(* Logix 5000 project; controller Transcat vendor 1 type 14 code 152 rev 32.11; software revision 32.02 *)

TASK MainTask (continuous, watchdog 500 ms) : MainProgram

MODULES
   Local : vendor 1 type 14 code 152 (PointIO 0, rev 32.11)
      MX201_LowerHowesVFD : PowerFlex 525-EENET (Ethernet 192.168.1.192, rev 5.1, Output RPI 20 ms)   // VFD for Lower Howes Mixer
           MX201_LowerHowesVFD:I.Ready   // LowerHowes Drive Ready Status
           MX201_LowerHowesVFD:I.Faulted   // LowerHowes Drive Faulted
           MX201_LowerHowesVFD:I.Active   // LowerHowes Drive Active
           MX201_LowerHowesVFD:O.Stop   // Drive Stop
      MX101_UpperHowesVFD : PowerFlex 525-EENET (Ethernet 192.168.1.191, rev 5.1, Output RPI 20 ms)   // VFD for Upper Howes Mixer
           MX101_UpperHowesVFD:I.Faulted   // UpperHowes Drive Faulted
           MX101_UpperHowesVFD:I.Active   // UpperHowes Drive Active
           MX101_UpperHowesVFD:I.Ready   // UpperHowes Drive Ready Status
           MX101_UpperHowesVFD:O.FreqCommand   // Input Hz into Source A: 0-60 Hz range
           MX101_UpperHowesVFD:O.Stop   // Drive Stop
           MX101_UpperHowesVFD:O.Start   // Drive Start
      VF101_Medium_Feeder : PowerFlex 525-EENET (Ethernet 192.168.1.193, rev 5.1, Output RPI 20 ms)   // Medium Feeder
      VF201_Small_Feeder_2 : PowerFlex 525-EENET (Ethernet 192.168.1.194, rev 5.1, Output RPI 20 ms)   // Small Feeder 2
      Thayer1_BS : ETHERNET-MODULE (Ethernet 192.168.1.140, rev 1.1, Output RPI 50 ms)   // Thayer 1 Weight Belt Feeder
      SBC2000_1_Acrison : ETHERNET-MODULE (Ethernet 192.168.1.150, rev 1.1, Output RPI 250 ms)   // Acrison Drive 1 to control Small Feeder 1
           SBC2000_1_Acrison:I.Data[1]   // PV - Feedrate - kg/hr
           SBC2000_1_Acrison:I.Data[2]   // Totalizer 1 - kg
           SBC2000_1_Acrison:I.Data[4]   // Hopper Level - %
           SBC2000_1_Acrison:I.Data[3]   // OT - Motor Speed - %
           SBC2000_1_Acrison:I.Data   // Ethernet Input Array
           SBC2000_1_Acrison:I.Data[0]   // SP-FeedRate - kg/hr
           SBC2000_1_Acrison:O.Data[15]   // When Command_Bits is 1, machine is running.
      Thayer2_BS : ETHERNET-MODULE (Ethernet 192.168.1.160, rev 1.1, Output RPI 50 ms)   // Thayer 2 Weigh Belt Feeder
      AENTPointIO : 1734-AENT (Ethernet 192.168.1.190, rev 3.1, Output RPI 20 ms)
         Slot1_420_8Input : vendor 1 type 115 code 210 (PointIO 1, rev 3.1, Input RPI 80 ms)
              AENTPointIO:1:I.Ch0Data   // LowerHowesSpeedSensorSignal
         Slot2_24V_8DI : 1734-IB8 (PointIO 2, rev 3.1)
      Discrete_IO : Embedded (PointIO 1, rev 32.11, Output RPI 20 ms)
           Local:1:O.Data.0   // Red Beacon Light
           Local:1:O.Data.3   // Blue Beacon Light
           Local:1:O.Data.1   // Yellow Beacon Light
           Local:1:O.Data.2   // Green Beacon Light
           Local:1:O.Data.4   // Beacon Buzzer/Sound
END_MODULES

TYPE Acrison_Feeder :   // Acrison Feeder Tags
STRUCT
   AutoMan : BOOL;   // On - Auto Control - follows AutoRun bit, Off - Manaul Control - follows Manual Run bit
   ManualRun : BOOL;   // On - Runs feeder in Manual, Off - Stops feeder in manual
   AutoRun : BOOL;   // On - Runs feeder in Auto Off - Stops feeder in Auto
   Interlock : BOOL;   // Interlock bit - if on - Feeder will not run
   Output : BOOL;   // On - Feeder runs, Off Feeder stops
   Int_Status : DINT;   // 32 Status bits from feeder
   SP_HMI : REAL;   // setpoint from HMI
   SP_READ : REAL;   // setpoint read back from controller
   Enable : BOOL;   // Enable logic to run feeder
   OT_Actual_Hz : REAL;   // The current output of the VFD in Hz
   FreqHz_Real : REAL;   // The command frequency of the drive in Hz
   CycleTime : TIMER;   // running time of current cycle
   CampTime : TIMER;   // running time of current campaign / batch
   TotalTime : TIMER;   // total time the device / motor has run since last reset
   OneShots : BOOL[32];   // 32 Booleans to hold one-shots assicated with this device
   TimeRunTarget : DINT;   // Target Amount of time in seconds to run the device
   StartDelay : TIMER;   // Delay before motor start
   StartDelayms : DINT;   // Start delay in milliseconds
   TimeRunStart : BOOL;   // Bit to start and run a timed run
END_STRUCT
END_TYPE

TYPE BronkhorstFlowMeter :   // Read and write values for Bronkhorst Flow Meters
STRUCT
   SP_R : REAL;   // Set Point - FlowRate - Read - g/min - read from Flow Meter
   PV_R : REAL;   // Process Variable - FlowRate - Read - g/min
   OT_R : REAL;   // Output - PumpSpeed - Read - %
   TempC : REAL;   // Temperaure - Read - Deg C
   Density : REAL;   // Density - Read - g/liter
   Usertag : STRING;   // User Tag in Flow Meter - String
   FBNode : INT;   // Flow Bus Node # - Integer
   Model : STRING;   // Flow Meter Model #
   Serial : STRING;   // Flow Meter Serial #
   Capacity : REAL;   // Max Flow Rate of Flow Meter
   Enable : BOOL;   // Device enable bit
   AutoMan : BOOL;   // Select Auto / Manual Mode
   AutoRun : BOOL;   // On / Off in Auto Mode
   ManualRun : BOOL;   // On / Off- in Manual Mode
   Interlock : BOOL;   // Interlock Bit
   Output : BOOL;   // Output Bit for Device
   SP_HMI : REAL;   // Setpoint from HMI
   SP_W : REAL;   // Setpoint - flowrate g/min - write to Flow Meter from PLC
   Connected : BOOL;   // Is flow meter connecte to the flow bus network
   Alarm : BOOL;   // Alarm Bit - if on flow meter in ALarm Status
   Running : BOOL;   // the flow meter is running / dosing
   AlarmReset : BOOL;   // bit to toggle to reset alarm
   AlarmID : INT;   // Integer # that describes the type of Alarm
   ReadTime : INT;   // time in milliseconds to read the flow meter data
   DevPct : REAL;   // % deviation of process variable from setpoint
   CycleTime : TIMER;   // running time of current cycle
   CampTime : TIMER;   // running time of current campaign
   TotalTime : TIMER;   // total time the device / motor has run since last reset
   OneShots : BOOL[32];   // 32 Booleans to hold one-shots assicated with this device
   TimeRunTarget : DINT;   // Target Amount of time in seconds to run the device
   StartDelay : TIMER;   // Delay before motor start
   StartDelayms : DINT;   // Start delay in milliseconds
   TimeRunStart : BOOL;   // Bit to start and run a timed run
   Totalizer : REAL;   // Total dosed by flow meter since last reset
   TotalizerReset : BOOL;   // Bit to reset the totalizer (called a counter in Bronkhorst literature)
END_STRUCT
END_TYPE

TYPE Howes_Mixer :   // Howes Mixer Tags
STRUCT
   AutoMan : BOOL;   // On - Auto Control - follows AutoRun bit, Off - Manaul Control - follows Manual Run bit
   ManualRun : BOOL;   // On - Runs feeder in Manual, Off - Stops feeder in manual
   AutoRun : BOOL;   // On - Runs feeder in Auto Off - Stops feeder in Auto
   Interlock : BOOL;   // Interlock bit - if on - Feeder will not run
   Output : BOOL;   // On - Feeder runs, Off Feeder stops
   Int_Status : DINT;   // 32 Status bits from feeder
   SP_HMI : REAL;   // setpoint from HMI
   SP_READ : REAL;   // setpoint read back from controller
   Enable : BOOL;   // Enable logic to run mixer
   FreqHz_Real : REAL;   // Frequency in Hz expressed as real #
   OT_Actual_Hz : REAL;   // The current output of the drive in Hz
   CycleTime : TIMER;   // currnet cycle run time
   CampTime : TIMER;   // current campaign run time
   TotalTime : TIMER;   // total run time since last reset
   OneShots : BOOL[32];   // 32 Booleans to hold one shots associated with this device
   TimeRunTarget : DINT;   // Target Amount of time in seconds to run the device
   TimeRunStart : BOOL;   // Bit to start and run a timed run
   StartDelay : TIMER;   // Delay before motor starts
   StartDelayms : DINT;   // Delay before motor starts in milliseconds
   RPM : REAL;   // RPM from speed sensor
END_STRUCT
END_TYPE

TYPE Thayer_WB_Feeder :   // Thayer WB Feeder Tags
STRUCT
   AutoMan : BOOL;   // On - Auto Control - follows AutoRun bit, Off - Manaul Control - follows Manual Run bit
   ManualRun : BOOL;   // On - Runs feeder in Manual, Off - Stops feeder in manual
   AutoRun : BOOL;   // On - Runs feeder in Auto Off - Stops feeder in Auto
   Interlock : BOOL;   // Interlock bit - if on - Feeder will not run
   Output : BOOL;   // On - Feeder runs, Off Feeder stops
   Int_Status : DINT;   // 32 Status bits from feeder
   SP_HMI : REAL;   // setpoint from HMI
   SP_READ : REAL;   // setpoint read back from controller
   Enable : BOOL;   // Enable logic to run feeder
   CycleTime : TIMER;   // current cycle run time
   CampTime : TIMER;   // current campaing run time
   TotalTime : TIMER;   // total run time since last reset
   OneShots : BOOL[32];   // 32 Booleans to hold one-shots assicated with this device
   TimeRunTarget : DINT;   // Target Amount of time in seconds to run the device - from recipe
   StartDelay : TIMER;   // Delay before starting motor / equipment
   StartDelayms : DINT;   // Start delay in milliseconds
   TimeRunStart : BOOL;   // Bit to start and run a timed run
END_STRUCT
END_TYPE

VAR_GLOBAL   (* controller tags *)
   AcrisonFeedRateSetPoint : MESSAGE;   // Message Command to Write to Feed Rate Set Point in Acrison from GF103.SP_HMI in kg/hr
        MessageParameters(ServiceCode := 16#0010, LocalElement := GF301.SP_HMI, ...)
   alwaysOFF : BOOL;
   BeaconBeepAlarm : ALIAS FOR Local:1:O.Data.4;   // Beep Alarm
   BeaconBlueLight : ALIAS FOR Local:1:O.Data.3;   // Blue Beacon Light
   BeaconGreenLight : ALIAS FOR Local:1:O.Data.2;   // Green Beacon Light
   BeaconRedLight : ALIAS FOR Local:1:O.Data.0;   // Red Beacon Light
   BeaconYellowLight : ALIAS FOR Local:1:O.Data.1;   // Yellow Beacon Light
   Beep : BOOL;   // Bit to Activte Beacon Alarm
   FT103 : BronkhorstFlowMeter := (PV_R := 8.803709, TempC := 22.585506, Density := 9999.0, Usertag := 'FT-103', Model := 'M55-RGD-25-0-S', Serial := 'M22213015A', Capacity := 1000.00006, Enable := 1, SP_HMI := 100.0, Connected := 1, ReadTime := 136, CycleTime.PRE := 288000000, CycleTime.ACC := 19487, CampTime.PRE := 28800000, CampTime.ACC := 10001, TotalTime.PRE := 999999999, TotalTime.ACC := 114629, Totalizer := 30.49);
   FT104 : BronkhorstFlowMeter := (PV_R := -9.60369, TempC := 22.258062, Density := 9999.0, Usertag := 'FT-104          ', Model := 'M55-RGD-25-0-S', Serial := 'M22213015C', Capacity := 10000.0, Enable := 1, SP_HMI := 100.0, Connected := 1, ReadTime := 80, CycleTime.PRE := 288000000, CycleTime.ACC := 3248, CampTime.PRE := 28800000, CampTime.ACC := 10001, TotalTime.PRE := 999999999, TotalTime.ACC := 84417, StartDelay.PRE := 2000, StartDelayms := 2, Totalizer := 6.64);
   FT105 : BronkhorstFlowMeter := (PV_R := 0.5630569, TempC := 29.962246, Density := 5.6385093, Usertag := 'FT-105          ', Model := 'M14-RGD-22-0-S', Serial := 'M20210127A', Capacity := 202.79999, Enable := 1, SP_HMI := 12.5, Connected := 1, ReadTime := 63, CycleTime.PRE := 288000000, CycleTime.ACC := 11357, CampTime.PRE := 28800000, CampTime.ACC := 10001, TotalTime.PRE := 999999999, TotalTime.ACC := 55929, StartDelay.PRE := 4000, StartDelayms := 4, Totalizer := 1840865.0);
   GF101 : Thayer_WB_Feeder := (SP_HMI := 10.0, SP_READ := 10.0, Enable := 1, CycleTime.PRE := 288000000, CycleTime.ACC := 9195, CampTime.PRE := 28800000, CampTime.ACC := 10001, TotalTime.PRE := 999999999, TotalTime.ACC := 1761327, StartDelay.PRE := 2000, StartDelayms := 2);   // Thayer 1 Tags
   GF101_Alarm_ExcessDevSP : ALIAS FOR Thayer1_BS:I.Data[8].7;   // Thayer 1 (GF101) - Alarm - excessive deviation from SP
   GF101_LoadCell : ALIAS FOR Thayer1Data[15];   // Thayer 1 (GF101) load cell in lbs
   GF101_LoadCellTempF : ALIAS FOR Thayer1Data[16];   // Thayer 1 (GF101) load cell temperature in Deg F
   GF101_OutputPct : ALIAS FOR Thayer1Data[5];   // Thayer 1 (GF101) Output to motor in pct - raw
   GF101_RunningLoad : ALIAS FOR Thayer1Data[0];   // Thayer 1 (GF101) Running Load - current load on belt in lbs
   GF101_RunningRate : ALIAS FOR Thayer1Data[1];   // Thayer 1 (GF101) Running Rate - current PV displayed on the operator screen
   GF101_RunningSpeed : ALIAS FOR Thayer1Data[2];   // Thayer 1 (GF101) Running Soeed - current speed of the belt in ft/min?
   GF101_SetPoint : ALIAS FOR Thayer1Data[3];   // Thayer 1 (GF101) SetPoint - in lb/min
   GF101_Shutdown_ExcessDevSp : ALIAS FOR Thayer1_BS:I.Data[10].7;   // Thayer 1 (GF101) - Shutdown - excessive deviation from SP
   GF101_Status_AutoMan : ALIAS FOR Thayer1_BS:I.Data[0].1;   // Thayer 1 (GF101) - Auto / Manual Status - 1 = Auto 0 = Manual
   GF101_Status_Coasting : ALIAS FOR Thayer1_BS:I.Data[0].2;   // Thayer 1 (GF101) - Coasting to stop of shutdown - 1 = Coasting, 0 = Not coasting
   GF101_Status_EchoBack : ALIAS FOR Thayer1_BS:I.Data[0].13;   // Thayer 1 (GF101) - Echo back bit
   GF101_Status_HeartBeat : ALIAS FOR Thayer1_BS:I.Data[0].14;   // Thayer 1 (GF101) - HeartBeat - every 5 seconds
   GF101_Status_Interlocked : ALIAS FOR Thayer1_BS:I.Data[0].8;   // Thayer 1 (GF101) - Interlocked Bit - 1 = Interlocked 0 = Not Interlocked
   GF101_Status_RunStop : ALIAS FOR Thayer1_BS:I.Data[0].0;   // Thayer 1 (GF101) - Operating Status - 1 = Running 0 = Stopped
   GF101_Status_TachGT0 : ALIAS FOR Thayer1_BS:I.Data[0].9;   // Thayer 1 (GF101) - 1 = Tachometer > 0 0 = Tachometer = 0
   GF101_TachHz : ALIAS FOR Thayer1Data[14];   // Thayer 1 (GF101) Tachometer in Hz
   GF101_Totalizer1 : ALIAS FOR Thayer1Data[9];   // Thayer 1 (GF101) Totalizer 1 in lbs
   GF101_Totalizer2 : ALIAS FOR Thayer1Data[10];   // Thayer 1 (GF101) Totalizer 2 in lbs
   GF101_Write_Acknowledge : ALIAS FOR Thayer1_BS:O.Data[2].5;   // Thayer 1 (GF101) Acknowledge
   GF101_Write_AutoMan : ALIAS FOR Thayer1_BS:O.Data[0].1;   // Thayer 1 (GF101) Auto / Manual 1 = Auto 2 = Manual
   GF101_Write_RunStop : ALIAS FOR Thayer1_BS:O.Data[0].0;   // Thayer 1 (GF101) 1 = Run / 0 = off/stop
   GF101_Write_Total1Reset : ALIAS FOR Thayer1_BS:O.Data[2].1;   // Thayer 1 (GF101) Totalizer 1 reset
   GF101_Write_Total2Reset : ALIAS FOR Thayer1_BS:O.Data[2].2;   // Thayer 1 (GF101) Totalizer 2 reset
   GF101OutpuyPct1sec : ALIAS FOR Thayer1Data[6];   // Thayer 1 (GF101) Output to motor in pct - averaged over 1 sec
   GF201 : Thayer_WB_Feeder := (SP_HMI := 5.0, SP_READ := 5.0, Enable := 1, CycleTime.PRE := 288000000, CycleTime.ACC := 17126, CampTime.PRE := 28800000, CampTime.ACC := 10001, TotalTime.PRE := 999999999, TotalTime.ACC := 1645614, StartDelay.PRE := 2000, StartDelayms := 2);   // Thayer 2 Tags
   GF201_Alarm_ExcessiDevSP : ALIAS FOR Thayer2_BS:I.Data[8].7;   // Thayer 2 (GF201) - Alarm - excessive deviation from SP
   GF201_LoadCell : ALIAS FOR Thayer2Data[15];   // Thayer 2 (GF201) load cell in lbs
   GF201_LoadCellTempF : ALIAS FOR Thayer2Data[16];   // Thayer 2 (GF201) load cell temperature in Deg F
   GF201_OutputPct : ALIAS FOR Thayer2Data[5];   // Thayer 2 (GF201) Output to motor in pct - raw
   GF201_RunningLoad : ALIAS FOR Thayer2Data[0];   // Thayer 2 (GF201) Running Load - current load on belt in lbs
   GF201_RunningRate : ALIAS FOR Thayer2Data[1];   // Thayer 2 (GF201) Running Rate - current PV displayed on the operator screen
   GF201_RunningSpeed : ALIAS FOR Thayer2Data[2];   // Thayer 2 (GF201) Running Soeed - current speed of the belt in ft/min?
   GF201_SetPoint : ALIAS FOR Thayer2Data[3];   // Thayer 2 (GF201) SetPoint - in lb/min
   GF201_Shutdown_ExcessDevSP : ALIAS FOR Thayer2_BS:I.Data[10].7;   // Thayer 2 (GF201) - Shutdown - excessive deviation from SP
   GF201_Status_AutoMan : ALIAS FOR Thayer2_BS:I.Data[0].1;   // Thayer 2 (GF201) - Auto / Manual Status - 1 = Auto 0 = Manual
   GF201_Status_Coasting : ALIAS FOR Thayer2_BS:I.Data[0].2;   // Thayer 2 (GF201) - Coasting to stop of shutdown - 1 = Coasting, 0 = Not coasting
   GF201_Status_EchoBack : ALIAS FOR Thayer2_BS:I.Data[0].13;   // Thayer 2 (GF201) - Echo back bit
   GF201_Status_HeartBeat1 : ALIAS FOR Thayer2_BS:I.Data[0].14;   // Thayer 2 (GF201) - HeartBeat - every 5 seconds
   GF201_Status_Interlocked : ALIAS FOR Thayer2_BS:I.Data[0].8;   // Thayer 2 (GF201) - Interlocked Bit - 1 = Interlocked 0 = Not Interlocked
   GF201_Status_RunStop : ALIAS FOR Thayer2_BS:I.Data[0].0;   // Thayer 2 (GF201) - Operating Status - 1 = Running 0 = Stopped
   GF201_Status_TachGT0 : ALIAS FOR Thayer2_BS:I.Data[0].9;   // Thayer 2 (GF201) - 1 = Tachometer > 0 0 = Tachometer = 0
   GF201_TachHz : ALIAS FOR Thayer2Data[14];   // Thayer 2 (GF201) Tachometer in Hz
   GF201_Totalizer1 : ALIAS FOR Thayer2Data[9];   // Thayer 2 (GF201) Totalizer 1 in lbs
   GF201_Totalizer2 : ALIAS FOR Thayer2Data[10];   // Thayer 2 (GF201) Totalizer 2 in lbs
   GF201_Write_Acknowledge : ALIAS FOR Thayer2_BS:O.Data[2].5;   // Thayer 2 (GF201) Acknowledge
   GF201_Write_AutoMan : ALIAS FOR Thayer2_BS:O.Data[0].1;   // Thayer 2 (GF201) Auto / Manual 1 = Auto 2 = Manual
   GF201_Write_Total1Reset : ALIAS FOR Thayer2_BS:O.Data[2].1;   // Thayer 2 (GF1201) Totalizer 1 reset
   GF201_Write_Total2Reset : ALIAS FOR Thayer2_BS:O.Data[2].2;   // Thayer 2 (GF201) Totalizer 2 reset
   GF201_Wrtie_RunStop : ALIAS FOR Thayer2_BS:O.Data[0].0;   // Thayer 2 (GF201) 1 = Run / 0 = off/stop
   GF201OutpuyPct1sec : ALIAS FOR Thayer2Data[6];   // Thayer 2 (GF201) Output to motor in pct - averaged over 1 sec
   GF301 : Acrison_Feeder := (Int_Status := 594012, SP_HMI := 6.7, Enable := 1, CycleTime.PRE := 288000000, CycleTime.ACC := 223848, CampTime.PRE := 28800000, CampTime.ACC := 10001, TotalTime.PRE := 999999999, TotalTime.ACC := 2086091, StartDelay.PRE := 2000, StartDelayms := 2);   // GF103 - Small Feeder 1
        .Int_Status.11   // Alarm
        .Int_Status.13   // Empty
        .Int_Status.10   // Overfill / Empty
        .Int_Status.3   // SP Int-1 / Ext-0
        .Int_Status   // 32 Bit Status Int
        .Int_Status.0   // Run-1 / Stop-0
        .Int_Status.5   // Batch-1 / Cont-0
        .Int_Status.4   // Mode - Grav-1 / Vol-0
        .Int_Status.6   // Batch Complete
        .Int_Status.1   // Refil
        .Int_Status.7   // Bribble
        .Int_Status.12   // Message
        .Int_Status.9   // Low Level
        .Int_Status.14   // Overfill
        .Int_Status.15   // Acrilock
        .Int_Status.16   // No Scale
        .Int_Status.17   // Deviation
        .Output   // GF103 - Acrison Small Feeder Run Bit
        .Int_Status.2   // AutoRefill
        .Int_Status.8   // High Level
   GF301_AlarmAck : BOOL;   // GF301 Alarm Ack Bit
   GF301_ClearCommands : BOOL;   // Bit to send clear command to GF301 command integer
   GF301_Command_Bits : INT;   // Command Word - Holds a value that gets written to Acrison SCB2000:I.Data[15] see Acrison Manual for which bits do what
        .0   // Run-1 / Stop-0
        .1   // Refill Mode Man - 1 / Auto - 0
        .2   // Batch-1 / Cont-0
        .3   // Batch Abort
        .4   // Refill ON
        .5   // Refill OFF
        .6   // Alarm Ack
        .7   // Mode Vol - 1/ Grav - 0
        .8   // Setpoint - Ext -1 / Int - 0
   GF301_IntStatus : DINT := 594012;   // 32 Bit Status INT for GF301
        .0   // Run- 1/ Stop - 0
        .1   // Refil
        .2   // Auto Refill
        .3   // Setpoint Int - 1 / Ext - 0
        .4   // Mode Grav - 1 / Vol - 0
        .5   // Batch - 1 / Cont - 0
        .6   // Batch Complete
        .7   // Dribble
        .8   // High Level
        .9   // Low Level
        .10   // Overfill / Empty
        .11   // Alarm
        .12   // Message
        .13   // Empty
        .14   // Overfill
        .15   // Acrilok
        .16   // No Scale
        .17   // Deviation
   GreenFlashingOff : TIMER := (PRE := 500);
   GreenFlashingOn : TIMER := (PRE := 500);
   HertzSetting : ALIAS FOR MX101_UpperHowesVFD:O.FreqCommand.0;   // UserHzSetting
   MSG_FROM_SLC500 : INT[10] := ([1] := 2500, [2] := 200, [3] := 300, [4] := 400, [5] := 500, [6] := 16, [7] := 17, [8] := 18, [9] := 19); {produced}
   MX101 : Howes_Mixer := (SP_HMI := 10.0, Enable := 1, FreqHz_Real := 6.0, CycleTime.PRE := 288000000, CycleTime.ACC := 4243, CampTime.PRE := 28800000, CampTime.ACC := 10001, TotalTime.PRE := 999999999, TotalTime.ACC := 1803981, StartDelay.PRE := 2000, StartDelayms := 2);
   MX201 : Howes_Mixer := (SP_HMI := 10.0, Enable := 1, FreqHz_Real := 6.0, CycleTime.PRE := 28800000, CycleTime.ACC := 117513, CampTime.PRE := 28800000, CampTime.ACC := 10001, TotalTime.PRE := 999999999, TotalTime.ACC := 1030054, StartDelay.PRE := 2000, StartDelayms := 2, RPM := -0.04);
   MX201_RPM_RAW : ALIAS FOR AENTPointIO:1:I.Ch3Data;   // Raw (unscaled) RMS reading from MX201 speed sensor - RPM * 100 (range 0 - 200 RPM)
   PowerOffThayer1 : BOOL;
   PowerOnThayer1 : BOOL;
   PT103_PV_RAW : ALIAS FOR AENTPointIO:1:I.Ch0Data;   // Raw (unscaled) pressure reading from PT103 - PSI * 100 (range 0 - 108 PSI)
   PT104_PV_RAW : ALIAS FOR AENTPointIO:1:I.Ch1Data;   // Raw (unscaled) pressure reading from PT104 - PSI * 100 (range 0 - 108 PSI)
   PT105_PV_RAW : ALIAS FOR AENTPointIO:1:I.Ch2Data;   // Raw (unscaled) pressure reading from PT105 - PSI * 100 (range 0 - 108 PSI)
   RandomFloat : REAL[20] := ([1] := 7.316811, [2] := 20.713356, [3] := 16.079597, [4] := 74.3938, [5] := 86.28061, [6] := 69.73996, [7] := 47.361, [8] := 43.876316, [9] := 89.62069, [10] := 56.526745);
   RecipeStart : BOOL;   // Bit to start and stop a recipe execution
   StartBeepTimer : TIMER := (PRE := 2500);   // Timer to sound the beep alarm before starting a device
   TempReal1 : REAL;
   Thayer1_SP : REAL := 20.0;
   Thayer1Ackn_SilenceRequest : BOOL;
   Thayer1Automatic : BOOL;
   Thayer1Data : REAL[40] := ([0] := 9.375, [1] := 3.109e-41, [3] := 10.0, [4] := 2.0, [9] := 1.5, [10] := 1.5046594, [11] := 5.4771e-41, [15] := 9.375, [16] := 70.66474, [17] := 1.6071e-41, [19] := 9.375);
        [10]   // Totalizer 2
        [3]   // SetPoint
        [2]   // Running Speed
        [0]   // Running Load
        [1]   // Running Rate
        [9]   // Totalizer 1
   Thayer1PowerOn : BOOL;
   Thayer1ResetTotalizers : BOOL;
   Thayer1SetPoint : REAL[1];
   Thayer1SpeedControl : REAL := 20.0;
   Thayer2_SP : REAL := 20.0;
   Thayer2Automatic : BOOL;
   Thayer2Data : REAL[40] := ([0] := 3.703125, [1] := 5.5868e-41, [3] := 5.0, [15] := 3.703125, [16] := 70.80019, [17] := 1.6071e-41, [19] := 3.703125);
   Thayer2PowerOn : BOOL;
   Thayer2ResetTotalizers : BOOL;
   Thayer2SpeedControl : REAL := 20.0;
   UHStartOneShot : BOOL;
   UHStopOneShot : BOOL;
   UpHowesHMIRun : BOOL;
   UpHowesHMIStop : BOOL;
   UpHowesSpeedHMI : INT;
   UpperHowesSpeed : INT := 2500;
   UpperHowesStart : BOOL;
   UpperHowesStop : BOOL;
   VF101 : Acrison_Feeder := (SP_HMI := 10.0, Enable := 1, FreqHz_Real := 6.0, CycleTime.PRE := 288000000, CycleTime.ACC := 7359, CampTime.PRE := 28800000, CampTime.ACC := 10001, TotalTime.PRE := 999999999, TotalTime.ACC := 1720239, StartDelay.PRE := 5000, StartDelayms := 5);   // Medium Feeder Tags
   VF201 : Acrison_Feeder := (SP_HMI := 10.0, Enable := 1, FreqHz_Real := 6.0, CycleTime.PRE := 288000000, CycleTime.ACC := 13534, CampTime.PRE := 28800000, CampTime.ACC := 10001, TotalTime.PRE := 999999999, TotalTime.ACC := 1964985, StartDelay.PRE := 5000, StartDelayms := 5);   // Small Feeder 2 Tags
   YellowFlashOff : TIMER := (PRE := 500);
   YellowFlashOn : TIMER := (PRE := 500, ACC := 180, EN := 1, TT := 1);
END_VAR

PROGRAM MainProgram   (* main routine MainRoutine *)
VAR
   AcrisonSpeedControl : REAL := 1.0;
   AcrisonSpeedControl2 : REAL := 15.0;
   HertzInput : INT := 20;
   Int_Status : DINT := 540252;
   LowerHowesSpeedSensor : REAL := -74.49097;
   PowerOffACrison : BOOL := 1;
   PowerOnAcrison : BOOL;
   SCL_01 : SCALE := (In := -3.0, InRawMax := 16384.0, InRawMin := 3271.0, InEUMax := 300.0, Out := -74.90277, MinAlarm := 1);
   SCL_02 : SCALE := (In := 16.0, InRawMax := 16384.0, InRawMin := 3271.0, InEUMax := 300.0, Out := -74.46809, MinAlarm := 1);
   SpeedSensorUpperHowesSpeed : REAL := -74.90277;
   T1 : TIMER := (PRE := 10000);
   T2 : TIMER := (PRE := 10000, ACC := 10000, EN := 1, DN := 1);
END_VAR

ROUTINE FT103_Oil_Dosing   (* ladder *)
// Logic to control FT103
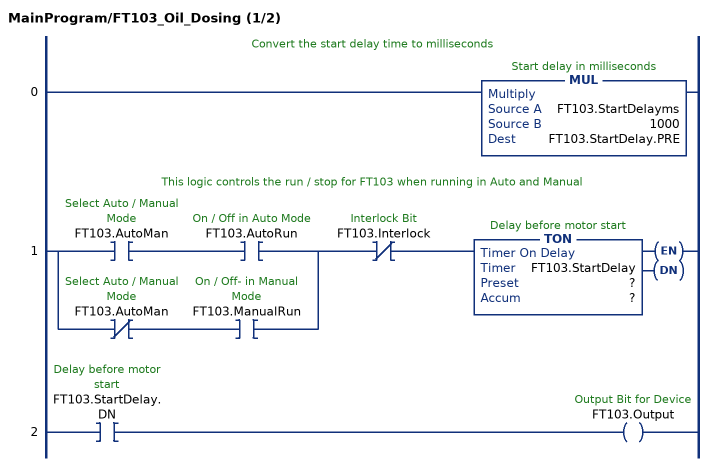
   // Convert the start delay time to milliseconds
   0: MUL(FT103.StartDelayms,1000,FT103.StartDelay.PRE);
   // This logic controls the run / stop for FT103 when running in Auto and Manual
   1: [XIC(FT103.AutoMan) XIC(FT103.AutoRun) ,XIO(FT103.AutoMan) XIC(FT103.ManualRun) ]XIO(FT103.Interlock)TON(FT103.StartDelay,?,?);
   2: XIC(FT103.StartDelay.DN)OTE(FT103.Output);
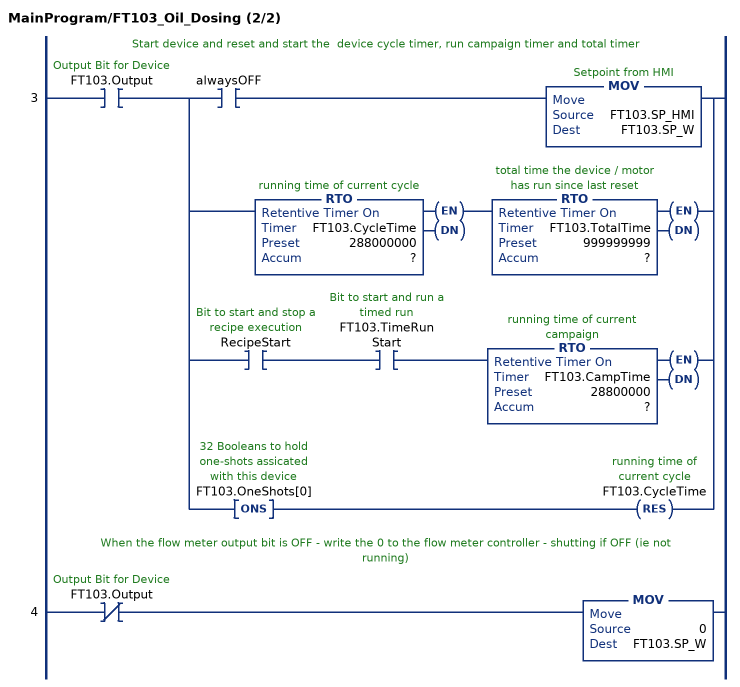
   // Start device and reset and start the  device cycle timer, run campaign timer and total timer
   3: XIC(FT103.Output)[XIC(alwaysOFF) MOV(FT103.SP_HMI,FT103.SP_W) ,[RTO(FT103.CycleTime,?,?) RTO(FT103.TotalTime,?,?) ,XIC(RecipeStart) XIC(FT103.TimeRunStart) RTO(FT103.CampTime,?,?) ,ONS(FT103.OneShots[0]) RES(FT103.CycleTime) ] ];
   // When the flow meter output bit is OFF - write the 0 to the flow meter controller - shutting if OFF (ie not running)
   4: XIO(FT103.Output)MOV(0,FT103.SP_W);
END_ROUTINE

ROUTINE FT104_Water_Dosing   (* ladder *)
// FT104 Control Logic
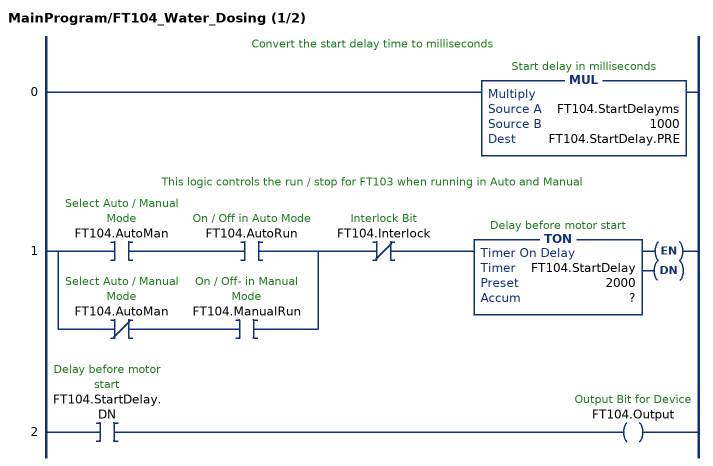
   // Convert the start delay time to milliseconds
   0: MUL(FT104.StartDelayms,1000,FT104.StartDelay.PRE);
   // This logic controls the run / stop for FT103 when running in Auto and Manual
   1: [XIC(FT104.AutoMan) XIC(FT104.AutoRun) ,XIO(FT104.AutoMan) XIC(FT104.ManualRun) ]XIO(FT104.Interlock)TON(FT104.StartDelay,?,?);
   2: XIC(FT104.StartDelay.DN)OTE(FT104.Output);
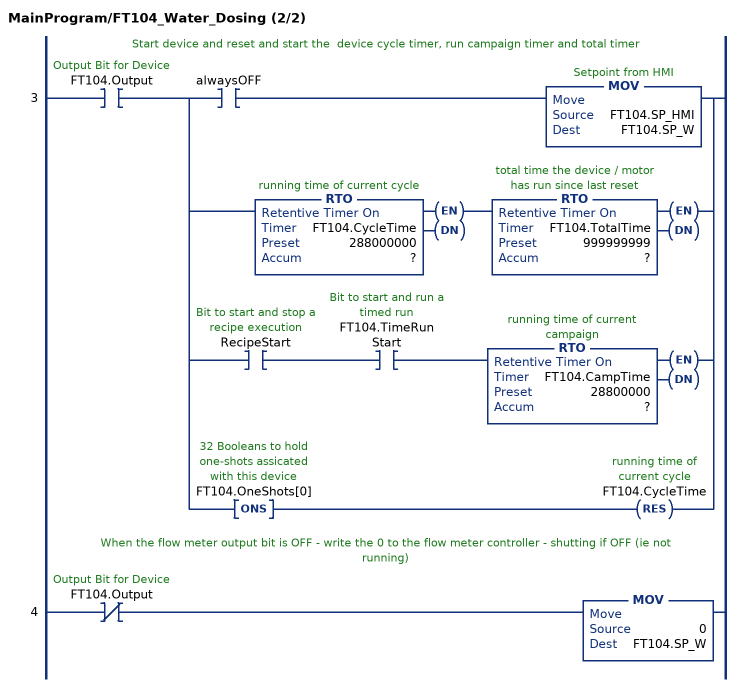
   // Start device and reset and start the  device cycle timer, run campaign timer and total timer
   3: XIC(FT104.Output)[XIC(alwaysOFF) MOV(FT104.SP_HMI,FT104.SP_W) ,[RTO(FT104.CycleTime,?,?) RTO(FT104.TotalTime,?,?) ,XIC(RecipeStart) XIC(FT104.TimeRunStart) RTO(FT104.CampTime,?,?) ,ONS(FT104.OneShots[0]) RES(FT104.CycleTime) ] ];
   // When the flow meter output bit is OFF - write the 0 to the flow meter controller - shutting if OFF (ie not running)
   4: XIO(FT104.Output)MOV(0,FT104.SP_W);
END_ROUTINE

ROUTINE FT105_Fragrance_Dosing   (* ladder *)
// FT105 Control Logic
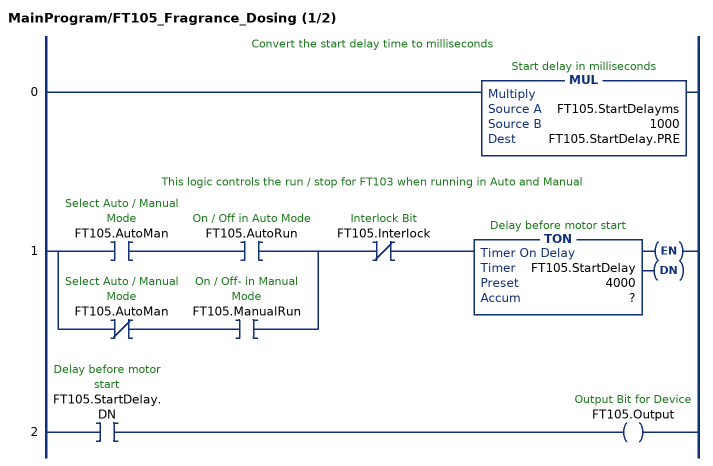
   // Convert the start delay time to milliseconds
   0: MUL(FT105.StartDelayms,1000,FT105.StartDelay.PRE);
   // This logic controls the run / stop for FT103 when running in Auto and Manual
   1: [XIC(FT105.AutoMan) XIC(FT105.AutoRun) ,XIO(FT105.AutoMan) XIC(FT105.ManualRun) ]XIO(FT105.Interlock)TON(FT105.StartDelay,?,?);
   2: XIC(FT105.StartDelay.DN)OTE(FT105.Output);
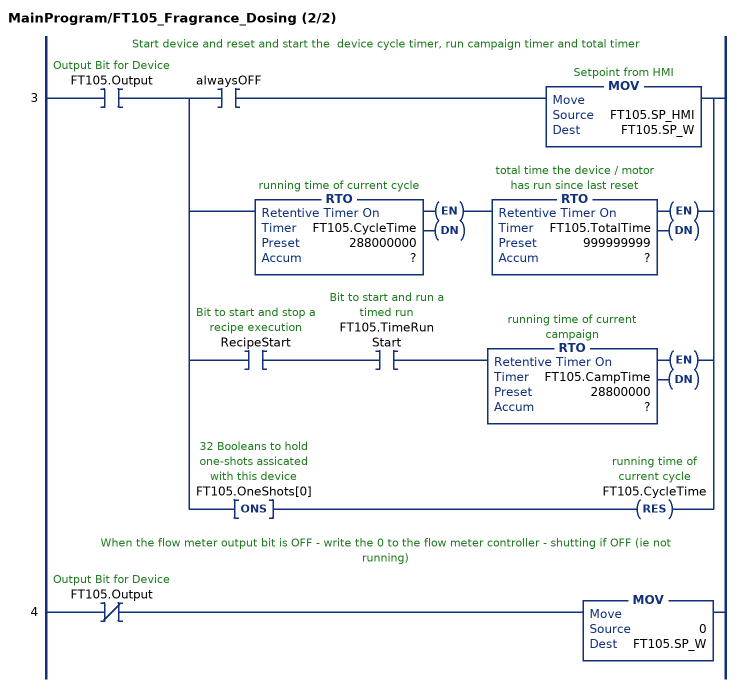
   // Start device and reset and start the  device cycle timer, run campaign timer and total timer
   3: XIC(FT105.Output)[XIC(alwaysOFF) MOV(FT105.SP_HMI,FT105.SP_W) ,[RTO(FT105.CycleTime,?,?) RTO(FT105.TotalTime,?,?) ,XIC(RecipeStart) XIC(FT105.TimeRunStart) RTO(FT105.CampTime,?,?) ,ONS(FT105.OneShots[0]) RES(FT105.CycleTime) ] ];
   // When the flow meter output bit is OFF - write the 0 to the flow meter controller - shutting if OFF (ie not running)
   4: XIO(FT105.Output)MOV(0,FT105.SP_W);
END_ROUTINE

ROUTINE GF101_Thayer1_WB_Feeder   (* ladder *)
// Thayer1 WB Feeder Control Logic (Old Limestone Feeder)
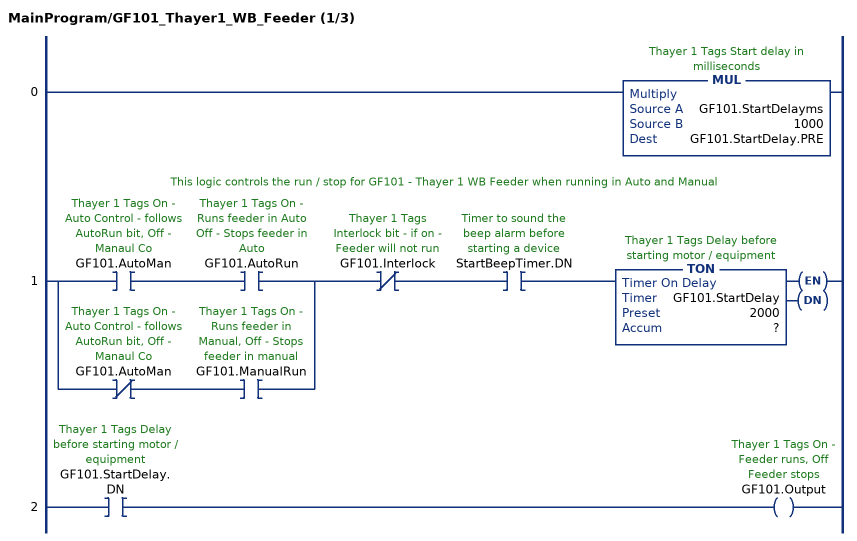
   0: MUL(GF101.StartDelayms,1000,GF101.StartDelay.PRE);
   // This logic controls the run / stop for GF101 - Thayer 1 WB Feeder when running in Auto and Manual
   1: [XIC(GF101.AutoMan) XIC(GF101.AutoRun) ,XIO(GF101.AutoMan) XIC(GF101.ManualRun) ]XIO(GF101.Interlock)XIC(StartBeepTimer.DN)TON(GF101.StartDelay,?,?);
   2: XIC(GF101.StartDelay.DN)OTE(GF101.Output);
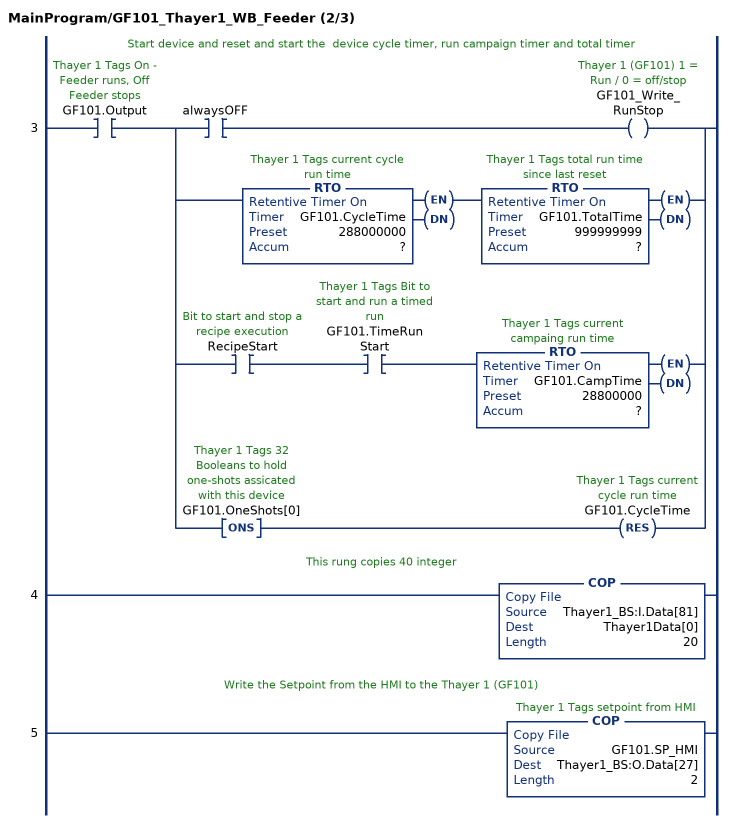
   // Start device and reset and start the  device cycle timer, run campaign timer and total timer
   3: XIC(GF101.Output)[XIC(alwaysOFF) OTE(GF101_Write_RunStop) ,[RTO(GF101.CycleTime,?,?) RTO(GF101.TotalTime,?,?) ,XIC(RecipeStart) XIC(GF101.TimeRunStart) RTO(GF101.CampTime,?,?) ,ONS(GF101.OneShots[0]) RES(GF101.CycleTime) ] ];
   // This rung copies 40 integer
   4: COP(Thayer1_BS:I.Data[81],Thayer1Data[0],20);
   // Write the Setpoint from the HMI to the Thayer 1 (GF101)
   5: COP(GF101.SP_HMI,Thayer1_BS:O.Data[27],2);
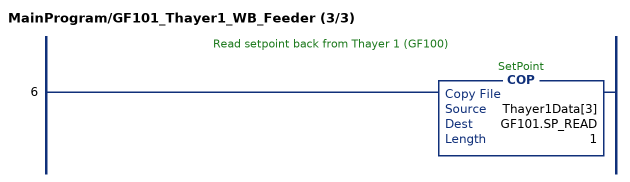
   // Read setpoint back from Thayer 1 (GF100)
   6: COP(Thayer1Data[3],GF101.SP_READ,1);
END_ROUTINE

ROUTINE GF201_Thayer2_WB_Feeder   (* ladder *)
// Thayer2 WB Feeder Control Logic (Old - Bentonite Feeder)
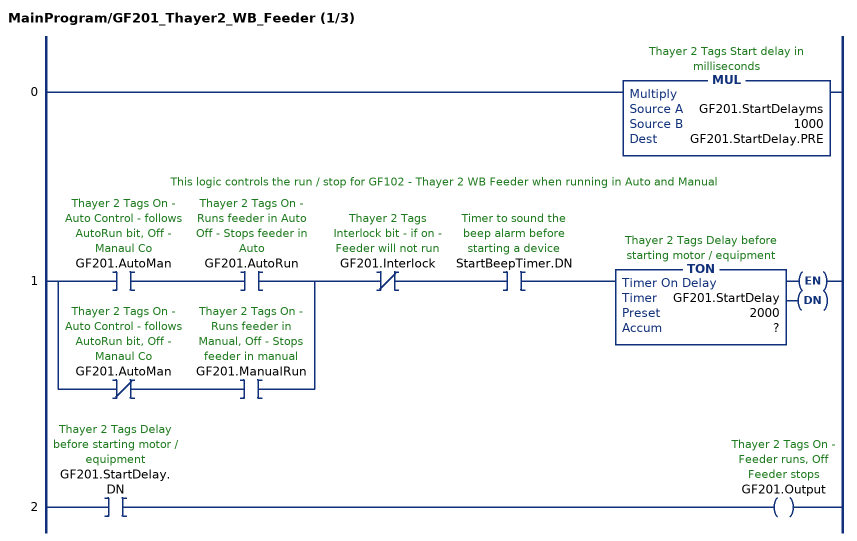
   0: MUL(GF201.StartDelayms,1000,GF201.StartDelay.PRE);
   // This logic controls the run / stop for GF102 - Thayer 2 WB Feeder when running in Auto and Manual
   1: [XIC(GF201.AutoMan) XIC(GF201.AutoRun) ,XIO(GF201.AutoMan) XIC(GF201.ManualRun) ]XIO(GF201.Interlock)XIC(StartBeepTimer.DN)TON(GF201.StartDelay,?,?);
   2: XIC(GF201.StartDelay.DN)OTE(GF201.Output);
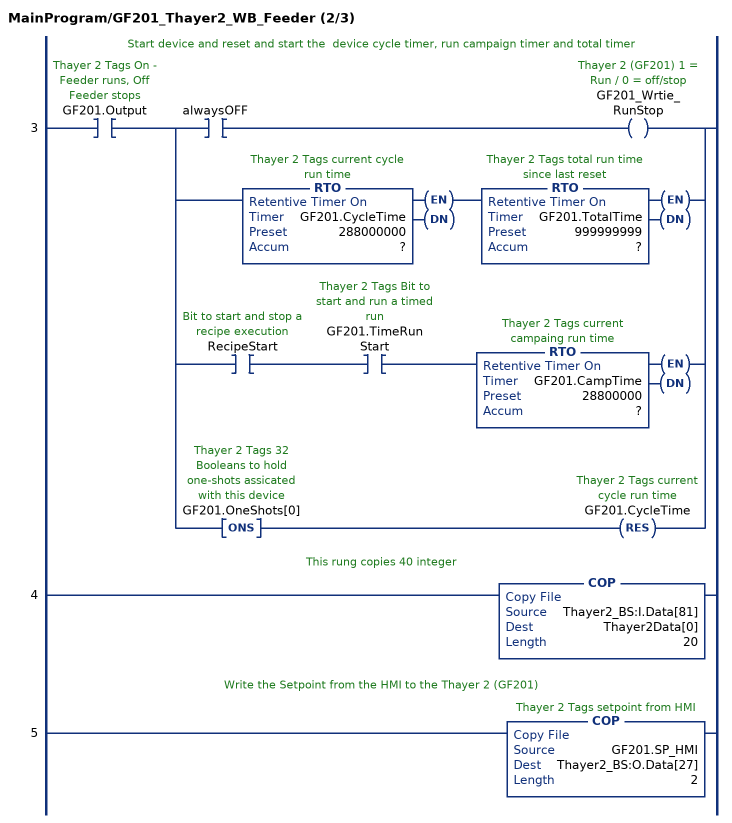
   // Start device and reset and start the  device cycle timer, run campaign timer and total timer
   3: XIC(GF201.Output)[XIC(alwaysOFF) OTE(GF201_Wrtie_RunStop) ,[RTO(GF201.CycleTime,?,?) RTO(GF201.TotalTime,?,?) ,XIC(RecipeStart) XIC(GF201.TimeRunStart) RTO(GF201.CampTime,?,?) ,ONS(GF201.OneShots[0]) RES(GF201.CycleTime) ] ];
   // This rung copies 40 integer
   4: COP(Thayer2_BS:I.Data[81],Thayer2Data[0],20);
   // Write the Setpoint from the HMI to the Thayer 2 (GF201)
   5: COP(GF201.SP_HMI,Thayer2_BS:O.Data[27],2);
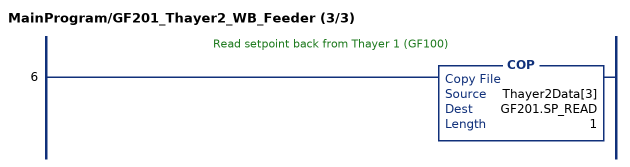
   // Read setpoint back from Thayer 1 (GF100)
   6: COP(Thayer2Data[3],GF201.SP_READ,1);
END_ROUTINE

ROUTINE GF301_Small_Feeder_AcrisonLIW   (* ladder *)
// Small Feeder 1 Control via Acrison Drive SBC 2000
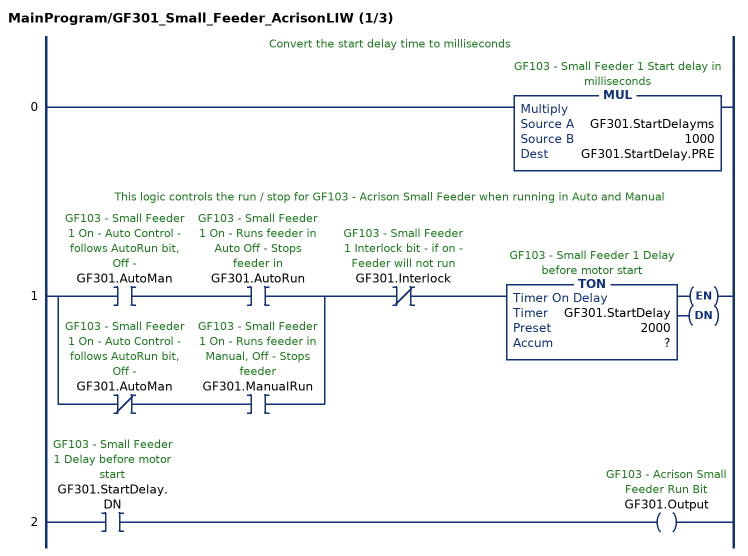
   // Convert the start delay time to milliseconds
   0: MUL(GF301.StartDelayms,1000,GF301.StartDelay.PRE);
   // This logic controls the run / stop for GF103 - Acrison Small Feeder when running in Auto and Manual
   1: [XIC(GF301.AutoMan) XIC(GF301.AutoRun) ,XIO(GF301.AutoMan) XIC(GF301.ManualRun) ]XIO(GF301.Interlock)TON(GF301.StartDelay,?,?);
   2: XIC(GF301.StartDelay.DN)OTE(GF301.Output);
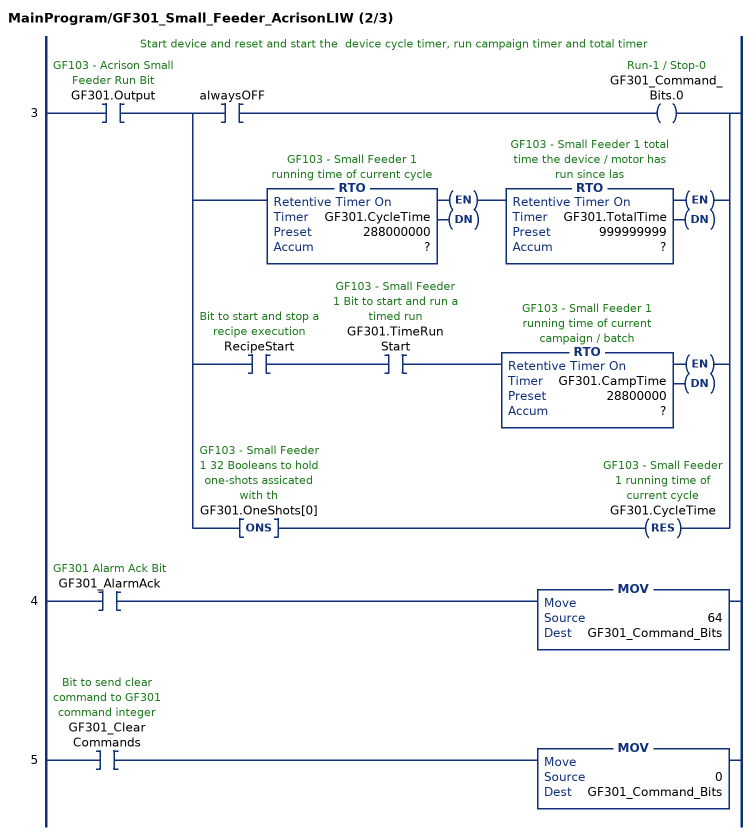
   // Start device and reset and start the  device cycle timer, run campaign timer and total timer
   3: XIC(GF301.Output)[XIC(alwaysOFF) OTE(GF301_Command_Bits.0) ,[RTO(GF301.CycleTime,?,?) RTO(GF301.TotalTime,?,?) ,XIC(RecipeStart) XIC(GF301.TimeRunStart) RTO(GF301.CampTime,?,?) ,ONS(GF301.OneShots[0]) RES(GF301.CycleTime) ] ];
   4: XIC(GF301_AlarmAck)MOV(64,GF301_Command_Bits);
   5: XIC(GF301_ClearCommands)MOV(0,GF301_Command_Bits);
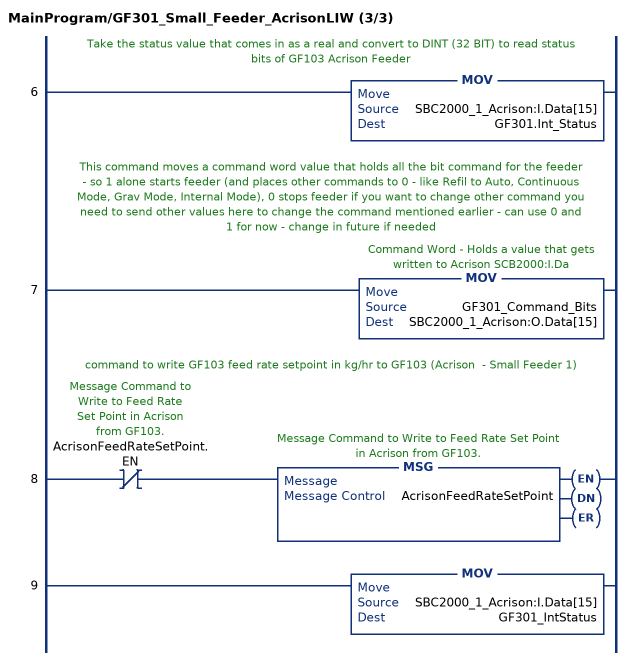
   // Take the status value that comes in as a real and convert to DINT (32 BIT) to read status bits of GF103 Acrison Feeder
   6: MOV(SBC2000_1_Acrison:I.Data[15],GF301.Int_Status);
   // This command moves a command word value that holds all the bit command for the feeder - so 1 alone starts feeder (and places other commands to 0 - like Refil to Auto, Continuous Mode, Grav Mode, Internal Mode), 0 stops feeder if you want to change other command you need to send other values here to change the command mentioned earlier - can use 0 and 1 for now - change in future if needed
   7: MOV(GF301_Command_Bits,SBC2000_1_Acrison:O.Data[15]);
   // command to write GF103 feed rate setpoint in kg/hr to GF103 (Acrison  - Small Feeder 1)
   8: XIO(AcrisonFeedRateSetPoint.EN)MSG(AcrisonFeedRateSetPoint);
   9: MOV(SBC2000_1_Acrison:I.Data[15],GF301_IntStatus);
END_ROUTINE

ROUTINE Light_Beacon   (* ladder *)
// Indicator Light Beacon
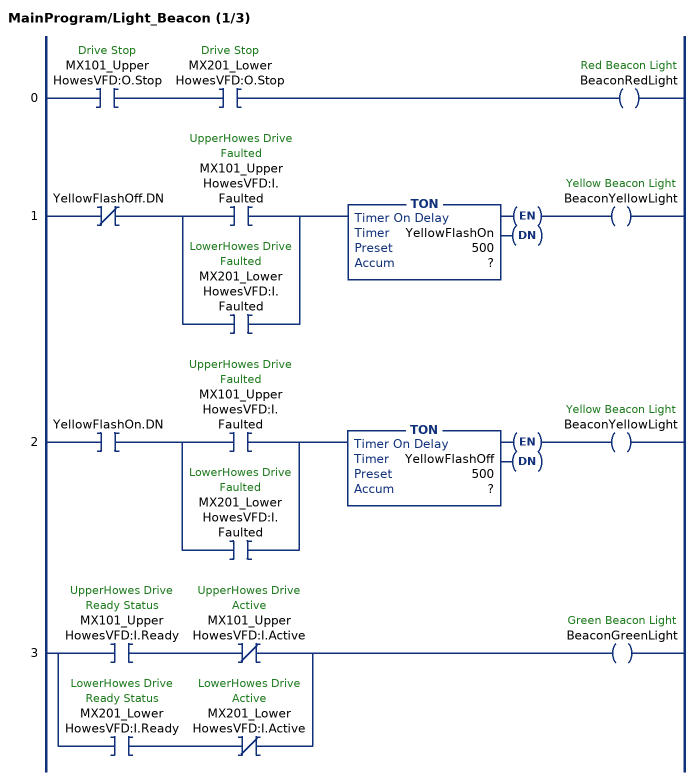
   0: XIC(MX101_UpperHowesVFD:O.Stop)XIC(MX201_LowerHowesVFD:O.Stop)OTE(BeaconRedLight);
   1: XIO(YellowFlashOff.DN)[XIC(MX101_UpperHowesVFD:I.Faulted) ,XIC(MX201_LowerHowesVFD:I.Faulted) ]TON(YellowFlashOn,?,?)OTE(BeaconYellowLight);
   2: XIC(YellowFlashOn.DN)[XIC(MX101_UpperHowesVFD:I.Faulted) ,XIC(MX201_LowerHowesVFD:I.Faulted) ]TON(YellowFlashOff,?,?)OTE(BeaconYellowLight);
   3: [XIC(MX101_UpperHowesVFD:I.Ready) XIO(MX101_UpperHowesVFD:I.Active) ,XIC(MX201_LowerHowesVFD:I.Ready) XIO(MX201_LowerHowesVFD:I.Active) ]OTE(BeaconGreenLight);
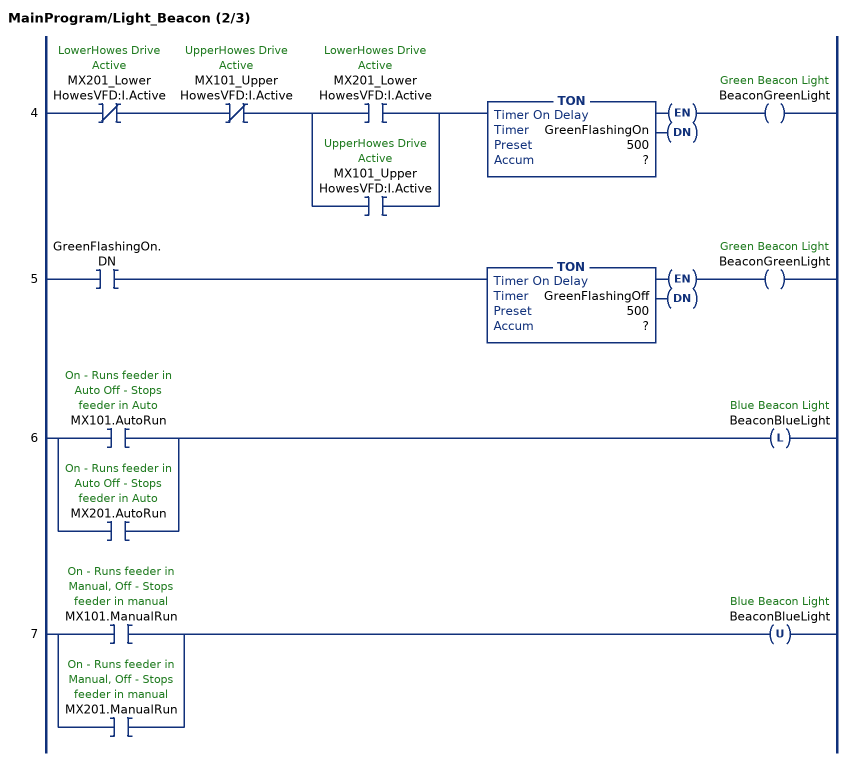
   4: XIO(MX201_LowerHowesVFD:I.Active)XIO(MX101_UpperHowesVFD:I.Active)[XIC(MX201_LowerHowesVFD:I.Active) ,XIC(MX101_UpperHowesVFD:I.Active) ]TON(GreenFlashingOn,?,?)OTE(BeaconGreenLight);
   5: XIC(GreenFlashingOn.DN)TON(GreenFlashingOff,?,?)OTE(BeaconGreenLight);
   6: [XIC(MX101.AutoRun) ,XIC(MX201.AutoRun) ]OTL(BeaconBlueLight);
   7: [XIC(MX101.ManualRun) ,XIC(MX201.ManualRun) ]OTU(BeaconBlueLight);
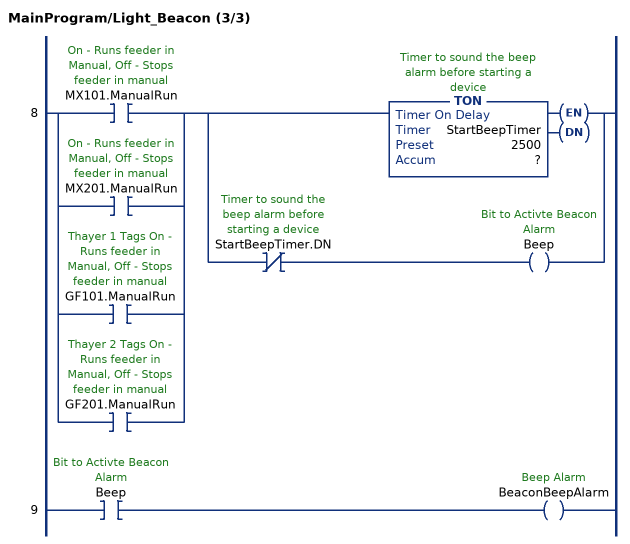
   8: [XIC(MX101.ManualRun) ,[XIC(MX201.ManualRun) ,[XIC(GF101.ManualRun) ,XIC(GF201.ManualRun) ] ] ][TON(StartBeepTimer,?,?) ,XIO(StartBeepTimer.DN) OTE(Beep) ];
   9: XIC(Beep)OTE(BeaconBeepAlarm);
END_ROUTINE
